Staubli VAL3: monitorAreaEn.dtx

public num nDistXCube[10]
public num nDistYCube[10]
public num nDistZCube[10]
public num nDistZCylinder[10]
public num nNumberCube = 9
public num nNumberCylinder = 9
public num nNumberFrame
public num nNumberSphere = 9
public num nRadiusCylinder[10]
public num nRadiusSphere[10]
  [9] = 600
public bool bCreateCube[10]
public bool bCreateCylinder[10]
bool bCreateFrame[10]
public bool bCreateSphere[10]
  [9] = true
frame fCube[10]
  [0] = {fatherId=world[0]}
  [1] = {fatherId=world[0]}
  [2] = {fatherId=world[0]}
  [3] = {fatherId=world[0]}
  [4] = {fatherId=world[0]}
  [5] = {fatherId=world[0]}
  [6] = {fatherId=world[0]}
  [7] = {fatherId=world[0]}
  [8] = {fatherId=world[0]}
  [9] = {fatherId=world[0]}
frame fCylinder[10]
  [0] = {fatherId=world[0]}
  [1] = {fatherId=world[0]}
  [2] = {fatherId=world[0]}
  [3] = {fatherId=world[0]}
  [4] = {fatherId=world[0]}
  [5] = {fatherId=world[0]}
  [6] = {fatherId=world[0]}
  [7] = {fatherId=world[0]}
  [8] = {fatherId=world[0]}
  [9] = {fatherId=world[0]}
frame fFrameZone[10]
  [0] = {fatherId=world[0]}
  [1] = {fatherId=world[0]}
  [2] = {fatherId=world[0]}
  [3] = {fatherId=world[0]}
  [4] = {fatherId=world[0]}
  [5] = {fatherId=world[0]}
  [6] = {fatherId=world[0]}
  [7] = {fatherId=world[0]}
  [8] = {fatherId=world[0]}
  [9] = {fatherId=world[0]}
frame fTableExample = {z=-50, fatherId=world[0]}
public pointRx pOriginCube[10]
  [0] = {fatherId=world[0]}
  [1] = {fatherId=world[0]}
  [2] = {fatherId=world[0]}
  [3] = {fatherId=world[0]}
  [4] = {fatherId=world[0]}
  [5] = {fatherId=world[0]}
  [6] = {fatherId=world[0]}
  [7] = {fatherId=world[0]}
  [8] = {fatherId=world[0]}
  [9] = {fatherId=world[0]}
public pointRx pOriginCylinder[10]
  [0] = {fatherId=world[0]}
  [1] = {fatherId=world[0]}
  [2] = {fatherId=world[0]}
  [3] = {fatherId=world[0]}
  [4] = {fatherId=world[0]}
  [5] = {fatherId=world[0]}
  [6] = {fatherId=world[0]}
  [7] = {fatherId=world[0]}
  [8] = {fatherId=world[0]}
  [9] = {fatherId=world[0]}
public pointRx pOriginSphere[10]
  [0] = {fatherId=world[0]}
  [1] = {fatherId=world[0]}
  [2] = {fatherId=world[0]}
  [3] = {fatherId=world[0]}
  [4] = {fatherId=world[0]}
  [5] = {fatherId=world[0]}
  [6] = {fatherId=world[0]}
  [7] = {fatherId=world[0]}
  [8] = {fatherId=world[0]}
  [9] = {y=300, z=1200, rx=180, fatherId=world[0]}
pointRx pStartExample = {x=400, z=100, fatherId=world[0]}
pointRx pStartExample2 = {x=600, z=-50, fatherId=world[0]}
